FUNCTION_BLOCK Actuator_StateOrder_subView
  (* Version 0.1, 2005-12-14, Oscar Ljungkrantz, Chalmers *)
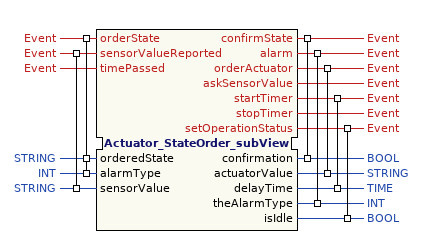
  EVENT_INPUT
    orderState WITH orderedState, alarmType;
    sensorValueReported WITH sensorValue;
    timePassed;
  END_EVENT
  EVENT_OUTPUT
    confirmState WITH confirmation;
    alarm WITH theAlarmType;
    orderActuator WITH actuatorValue;
    askSensorValue;
    startTimer WITH delayTime;
    stopTimer;
    setOperationStatus WITH isIdle;
  END_EVENT
  VAR_INPUT
    orderedState : STRING;
    alarmType : INT;
    sensorValue : STRING;
  END_VAR
  VAR_OUTPUT
    confirmation : BOOL;
    actuatorValue : STRING;
    delayTime : TIME;
    theAlarmType : INT;
    isIdle : BOOL;
  END_VAR
  VAR
    currentOrderedState : STRING;
    currentAlarmType : INT := 1;
    time : TIME := T#1h;
    operating : BOOL := FALSE;
  END_VAR
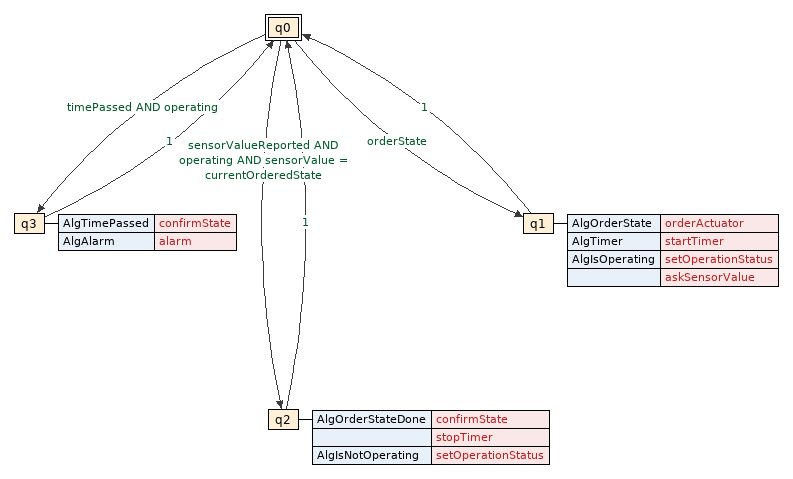
  EC_STATES
    q0;
    q1 : AlgOrderState -> orderActuator, AlgTimer -> startTimer, AlgIsOperating -> setOperationStatus, -> askSensorValue;
    q2 : AlgOrderStateDone -> confirmState, -> stopTimer, AlgIsNotOperating -> setOperationStatus;
    q3 : AlgTimePassed -> confirmState, AlgAlarm -> alarm;
  END_STATES
  EC_TRANSITIONS
    q0 TO q1 := orderState;
    q1 TO q0 := 1;
    q0 TO q2 := sensorValueReported AND operating AND sensorValue = currentOrderedState;
    q2 TO q0 := 1;
    q0 TO q3 := timePassed AND operating;
    q3 TO q0 := 1;
  END_TRANSITIONS
  ALGORITHM AlgOrderState IN Java:
		currentOrderedState = orderedState;
		currentAlarmType = alarmType;
		actuatorValue = currentOrderedState;
  END_ALGORITHM
  ALGORITHM AlgTimer IN Java:
		delayTime = time;
  END_ALGORITHM
  ALGORITHM IsOperating IN Java:
		isIdle = FALSE;
		operating = TRUE;
  END_ALGORITHM
  ALGORITHM AlgOrderStateDone IN Java:
		confirmation = TRUE;
  END_ALGORITHM
  ALGORITHM AlgIsNotOperating IN Java:
		isIdle = TRUE;
		operating = FALSE;
  END_ALGORITHM
  ALGORITHM AlgTimePassed IN Java:
		confirmation = FALSE;
  END_ALGORITHM
  ALGORITHM AlgAlarm IN Java:
		theAlarmType = currentAlarmType;
  END_ALGORITHM
END_FUNCTION_BLOCK
